INTERFACE I_HumiditySensor

PROPERTY Humidity : REAL
GET
END_GET
END_PROPERTY

END_INTERFACE

(* stored: Version 1.1.0.1
   Itf I_HumiditySensor: Id {46ec89d5-3c5f-466c-85ba-d291fb8e6f47}
   Property Humidity: Id {ea77c722-472d-406a-a74a-01de788c3ffc}
   Get Get: Id {1d6d4099-5682-4aa7-ae14-68f1f759aaca} *)
